Fanuc TP program (LS listing): _retreat_grind.ls

/PROG  _RETREAT_GRIND
/ATTR
OWNER		= MNEDITOR;
COMMENT		= "";
PROG_SIZE	= 275;
CREATE		= DATE 21-08-19  TIME 21:16:16;
MODIFIED	= DATE 21-08-19  TIME 21:16:16;
FILE_NAME	= RETREAT_;
VERSION		= 0;
LINE_COUNT	= 4;
MEMORY_SIZE	= 631;
PROTECT		= READ_WRITE;
TCD:  STACK_SIZE	= 0,
      TASK_PRIORITY	= 50,
      TIME_SLICE	= 0,
      BUSY_LAMP_OFF	= 0,
      ABORT_REQUEST	= 0,
      PAUSE_REQUEST	= 0;
DEFAULT_GROUP	= 1,*,*,*,*;
CONTROL_CODE	= 00000000 00000000;
/APPL
/APPL

AUTO_SINGULARITY_HEADER;
  ENABLE_SINGULARITY_AVOIDANCE   : TRUE;
/MN
   1:  PR[3:WELD OFFSET]=LPOS    ;
   2:  PR[3,3:WELD OFFSET]=(R[100:RETREAT]) ;
   3:  PR[3,5:WELD OFFSET]=(10) ;
   4:J PR[3:WELD OFFSET] 100% CNT10    ;
/POS
/END
